FUNCTION_BLOCK T_AsyncCommand IMPLEMENTS I_AsyncStatus
VAR
	_busy : BOOL;
	_done : BOOL;
	_error : BOOL;
END_VAR

{warning 'add property implementation'}
PROPERTY Busy : BOOL
GET
END_GET
END_PROPERTY

{warning 'add property implementation'}
PROPERTY Done : BOOL
GET
END_GET
END_PROPERTY

{warning 'add property implementation'}
PROPERTY Error : BOOL
GET
END_GET
END_PROPERTY

METHOD SetBusy : BOOL
VAR_INPUT
END_VAR
_busy := TRUE;
_done := FALSE;
_error := false;
END_METHOD

METHOD SetDone : BOOL
VAR_INPUT
END_VAR
_done := TRUE;
_error := FALSE;
_busy := false;
END_METHOD

METHOD SetError : BOOL
VAR_INPUT
END_VAR
_error := TRUE;
_done := FALSE;
_busy := false;
END_METHOD

END_FUNCTION_BLOCK

(* stored: Version 1.1.0.1, ProductVersion 3.1.4024.3
   POU T_AsyncCommand: Id {f43e4fe5-c7e6-4e3a-91bc-4289e77e3004}, SpecialFunc None
   Property Busy: Id {8fec2c7b-c104-4b70-ad59-4160bffd4620}
   Get Get: Id {b235158b-775b-47f4-ba67-c7d41c97db6d}
   Property Done: Id {04c9b1c1-a215-43b5-a97a-da57ffbd1460}
   Get Get: Id {d158fd72-60de-46f8-8c7f-a43a58c79538}
   Property Error: Id {2da61391-b887-42c2-9f86-c028099adb31}
   Get Get: Id {66d0aa16-ff42-4844-bc9d-5e8dfc692797}
   Method SetBusy: Id {31d01a92-ef17-4667-b6a2-907df7a7a2ee}
   Method SetDone: Id {9d386a3b-54a5-4fe5-a469-e8514beaca48}
   Method SetError: Id {8efea276-9126-4129-851d-1b356128b3c3} *)
